{attribute 'GeneratedUsingTerminal: EK1521-0010-0020'}
{attribute addProperty BoxType "EK1521-0010-0020"}
{attribute addProperty Id "InfoDataAT %I*InfoData_6F19DB2B2"}
{attribute addProperty CRC "532711307"}
{attribute addProperty Size "2"}
TYPE EK1521_1FC0878B EXTENDS EtcSlaveTerminalBase_947E5A46 :
STRUCT
	{attribute addProperty Name "InfoData"}
	InfoData : InfoData_6F19DB2B;
END_STRUCT
END_TYPE

(* stored: Version 1.2.0.0, ProductVersion 3.1.4024.9
   DUT EK1521_1FC0878B: Id {bcd64046-32b2-415e-9127-728a5843d841} *)
